FUNCTION_BLOCK INTERNAL FB_DirectoryUtilities_Tests EXTENDS FB_TestSuite
VAR_INPUT
END_VAR
VAR_OUTPUT
END_VAR
VAR
	_directoryUtilities	: FB_DirectoryUtilities;
END_VAR

Test01_CreateFile_Wait3Seconds_DeleteWithFileCreatedBeforeMethod();
Test02_TryDeletingButNoFilesMatchCriteria_ExpectNoErrors();

METHOD Test01_CreateFile_Wait3Seconds_DeleteWithFileCreatedBeforeMethod
VAR_INPUT
END_VAR
VAR_INST
	fileCreated			: BOOL;
	delayForDelete		: Tc2_Standard.TON;
	currentSystemTime	: DT;
	getSystemTime		: Tc2_System.GETSYSTEMTIME;
	fileTime			: Tc2_Utilities.T_FILETIME;
	dateTime			: DT;
	dtUpperLimit  		: DT  := DATE_AND_TIME#2106-02-07-06:28:15;
	error				: BOOL;
	errorInfo			: ZigaLibs_Core.ST_AdsError;
	deletedFiles		: ARRAY[0..100] OF Tc2_System.T_MaxString;
END_VAR
IF TcUnit.TEST_ORDERED('Test01_CreateFile_Wait3Seconds_DeleteWithFileCreatedBeforeMethod') THEN
	IF NOT fileCreated THEN
		IF Utilities.File.Create(PRG_TESTS.FILE_HANDLER_TESTS_PATH, 'FileToDeleteViaDeleteBeforeMethod.txt', '', FALSE, 
			error => error ,errorInfo => errorInfo)
		THEN
			fileCreated := TRUE;
			AssertFalse(error, Tc2_Standard.CONCAT('Unexpected error when creating the file: ', errorInfo.Message));
		END_IF
	ELSE
		delayForDelete(IN := TRUE, PT := T#3S);
		IF delayForDelete.Q THEN
			getSystemTime(timeHiDW => fileTime.dwHighDateTime, timeLoDW => fileTime.dwLowDateTime);
			IF _directoryUtilities.DeleteFilesCreatedBefore(PRG_TESTS.FILE_HANDLER_TESTS_PATH, 'FileToDeleteViaDeleteBeforeMet', '', dtUpperLimit, 
				error=> error, errorInfo => errorInfo, deletedFiles => deletedFiles)
			THEN
				AssertTrue(deletedFiles[0] = 'FileToDeleteViaDeleteBeforeMethod.txt', 'Deleted files list contains no items!');
				AssertFalse(error, Tc2_Standard.CONCAT('Deleting files encountered an undexpected error: ', errorInfo.Message));
				TcUnit.TEST_FINISHED();
			END_IF
		END_IF
	END_IF
END_IF
END_METHOD

METHOD Test02_TryDeletingButNoFilesMatchCriteria_ExpectNoErrors
VAR_INPUT
END_VAR
VAR_INST
	fileTime			: Tc2_Utilities.T_FILETIME;
	dateTime			: DT;
	dtUpperLimit  		: DT  := DATE_AND_TIME#2106-02-07-06:28:15;
	error				: BOOL;
	errorInfo			: ZigaLibs_Core.ST_AdsError;
	deletedFiles		: ARRAY[0..100] OF Tc2_System.T_MaxString;
END_VAR
IF TcUnit.TEST_ORDERED('Test02_TryDeletingButNoFilesMatchCriteria_ExpectNoErrors') THEN
	IF Utilities.Directory.DeleteFilesCreatedBefore(PRG_TESTS.FILE_HANDLER_TESTS_PATH, 'MyLog', PRG_TESTS.NET_ID, dtUpperLimit, 
				error=> error, errorInfo => errorInfo, deletedFiles => deletedFiles) THEN
	AssertFalse(error, 'An error has happened attempting to call the DeleteFilesCreatedBefore with no matching content provided.');
	TcUnit.TEST_FINISHED();
	END_IF
END_IF
END_METHOD

END_FUNCTION_BLOCK

(* stored: Version 1.1.0.1, ProductVersion 3.1.4024.15
   POU FB_DirectoryUtilities_Tests: Id {ed7d6ffd-1136-0ce4-3b13-cdf20f3d89ea}, SpecialFunc None
   Method Test01_CreateFile_Wait3Seconds_DeleteWithFileCreatedBeforeMethod: Id {52a00fe1-3600-0e91-2c94-bc06e7c79de6}
   Method Test02_TryDeletingButNoFilesMatchCriteria_ExpectNoErrors: Id {a96f2f3c-9905-0d39-3a55-66f90cf0cc77} *)
